# EPICS substitutions: siteApps/Example-1-2/alarmApp/Db/alarmEx.substitutions
file db/alarmEx.db {
  pattern { n }
    { 1 }
    { 2 }
    { 3 }
    { 4 }
    { 5 }
    { 6 }
    { 7 }
    { 8 }
    { 9 }
    { 10 }
}
